{attribute 'linkalways'} 
{attribute 'no_explicit_call' := 'This FB is a CLASS and must be accessed using methods or properties'}
{attribute 'enable_dynamic_creation'}
FUNCTION_BLOCK _TIMESTRUCT EXTENDS StructuredDatatypeBase
VAR
	localData : TIMESTRUCT;
	activeData : REFERENCE TO TIMESTRUCT REF= localData;
	_wYear : _WORD(localData.wYear);
	_wMonth : _WORD(localData.wMonth);
	_wDayOfWeek : _WORD(localData.wDayOfWeek);
	_wDay : _WORD(localData.wDay);
	_wHour : _WORD(localData.wHour);
	_wMinute : _WORD(localData.wMinute);
	_wSecond : _WORD(localData.wSecond);
	_wMilliseconds : _WORD(localData.wMilliseconds);
END_VAR

PROPERTY PUBLIC Address : PVOID
GET
Address := ADR(activeData);
END_GET
END_PROPERTY

METHOD PUBLIC ClearReference
VAR_INPUT
END_VAR
activeData REF= localData;
SetMemberReference();
END_METHOD

METHOD PUBLIC Clone : I_Datatype
VAR
    pClone : POINTER TO _TIMESTRUCT;
END_VAR
pClone := __NEW(_TIMESTRUCT());
pClone^.Value := Value;
Clone := pClone^;
END_METHOD

METHOD FB_init : BOOL
VAR_INPUT
	bInitRetains : BOOL; // if TRUE, the retain variables are initialized (warm start / cold start)
	bInCopyCode : BOOL;  // if TRUE, the instance afterwards gets moved into the copy code (online change)
END_VAR
SetMemberReference();
AddMember('wYear',_wYear);
AddMember('wMonth',_wMonth);
AddMember('wDayOfWeek',_wDayOfWeek);
AddMember('wDay',_wDay);
AddMember('wHour',_wHour);
AddMember('wMinute',_wMinute);
AddMember('wSecond',_wSecond);
AddMember('wMilliseconds',_wMilliseconds);
END_METHOD

PROPERTY PUBLIC Identifier : T_MAXSTRING
GET
Identifier := 'TIMESTRUCT';
END_GET
END_PROPERTY

METHOD PUBLIC MakeReferenceTo
VAR_INPUT
	ReferenceTarget : REFERENCE TO TIMESTRUCT;
END_VAR
activeData REF= ReferenceTarget;
SetMemberReference();
END_METHOD

METHOD PROTECTED SetMemberReference
VAR_INPUT
END_VAR
_wYear.MakeReferenceTo(activeData.wYear);
_wMonth.MakeReferenceTo(activeData.wMonth);
_wDayOfWeek.MakeReferenceTo(activeData.wDayOfWeek);
_wDay.MakeReferenceTo(activeData.wDay);
_wHour.MakeReferenceTo(activeData.wHour);
_wMinute.MakeReferenceTo(activeData.wMinute);
_wSecond.MakeReferenceTo(activeData.wSecond);
_wMilliseconds.MakeReferenceTo(activeData.wMilliseconds);
END_METHOD

PROPERTY PUBLIC Size : UDINT
GET
Size := SIZEOF(activeData);
END_GET
END_PROPERTY

METHOD TryMakeReferenceTo : BOOL
VAR_INPUT
	Target : I_Datatype;
END_VAR
VAR
	pTargetData : POINTER TO TIMESTRUCT;
END_VAR
IF NOT (Target.TypeName = TypeName) THEN
	RETURN;
END_IF

pTargetData := Target.Address;
activeData REF= pTargetData^;
SetMemberReference();
TryMakeReferenceTo := TRUE;
END_METHOD

PROPERTY PUBLIC Value : REFERENCE TO TIMESTRUCT
GET
Value REF= activeData;
END_GET
END_PROPERTY

PROPERTY PUBLIC wDay : Reference to _WORD
GET
wDay REF= _wDay;
END_GET
END_PROPERTY

PROPERTY PUBLIC wDayOfWeek : Reference to _WORD
GET
wDayOfWeek REF= _wDayOfWeek;
END_GET
END_PROPERTY

PROPERTY PUBLIC wHour : Reference to _WORD
GET
wHour REF= _wHour;
END_GET
END_PROPERTY

PROPERTY PUBLIC wMilliseconds : Reference to _WORD
GET
wMilliseconds REF= _wMilliseconds;
END_GET
END_PROPERTY

PROPERTY PUBLIC wMinute : Reference to _WORD
GET
wMinute REF= _wMinute;
END_GET
END_PROPERTY

PROPERTY PUBLIC wMonth : Reference to _WORD
GET
wMonth REF= _wMonth;
END_GET
END_PROPERTY

PROPERTY PUBLIC wSecond : Reference to _WORD
GET
wSecond REF= _wSecond;
END_GET
END_PROPERTY

PROPERTY PUBLIC wYear : Reference to _WORD
GET
wYear REF= _wYear;
END_GET
END_PROPERTY

END_FUNCTION_BLOCK

(* stored: Version 1.1.0.1, ProductVersion 3.1.4024.12
   POU _TIMESTRUCT: Id {e562b4d5-1171-0283-3cd5-573928ea5f08}, SpecialFunc None
   Folder Constructor: Id {a76fe964-4813-0dcc-3a87-52590a5beee4}
   Folder Protected: Id {b9713e34-49dc-0c25-27b9-d826f124e7e3}
   Property Address: Id {bb392fc3-3f0a-0e40-3700-c5663ef20063}
   Get Get: Id {6c22c66d-e36f-0aa4-2e36-5137ed472e2a}
   Method ClearReference: Id {2cb1a7a5-525f-094b-192a-13a283037e83}
   Method Clone: Id {351d97c3-851a-0daa-253f-1e9867ba5cc1}
   Method FB_init: Id {de249045-14c0-0c8e-3c32-9e332517c285}
   Property Identifier: Id {320cbb58-8004-0152-2111-dbc950bf6d4d}
   Get Get: Id {22f478c1-48ff-0d8c-1e28-359278e8bec7}
   Method MakeReferenceTo: Id {212e5344-3a4d-0d8c-22d5-17c348eff1df}
   Method SetMemberReference: Id {153ff1cd-4750-0dd7-22e7-155c91555b63}
   Property Size: Id {212b9de1-90be-01f3-0673-9ded294ddc75}
   Get Get: Id {541f10ed-fb82-0760-3537-2ccba0ff1404}
   Method TryMakeReferenceTo: Id {436cbb68-52af-07f8-1875-c0f6af217281}
   Property Value: Id {aae5b600-b6e3-0a73-2071-e343a31d09f7}
   Get Get: Id {595b6fc1-b502-08e3-2f56-be28310fd013}
   Property wDay: Id {bdfde783-bbe0-0f05-2fda-747386cce035}
   Get Get: Id {2ff1f2ca-f10f-022c-12ce-cb56c90848c2}
   Property wDayOfWeek: Id {b3a7e28e-5e16-0746-0099-3fb50c70e777}
   Get Get: Id {f945a899-5b24-0781-3fef-24a9bc7b1ba0}
   Property wHour: Id {91565ed2-d330-0a7e-029e-facc5a7353e9}
   Get Get: Id {0672e413-fccd-0ef3-08cb-16aef2b34fd1}
   Property wMilliseconds: Id {9bf32d92-8c98-07f4-25c8-2d263c2e8511}
   Get Get: Id {ae5e8915-e489-039a-29fa-4de80ddbf57b}
   Property wMinute: Id {eed4cd1f-750b-0370-146a-dd8fe50b813b}
   Get Get: Id {4e73a3f3-2a8c-07c4-18aa-47c3230d9fee}
   Property wMonth: Id {d96efd92-1a68-076b-05e4-58cd4947e090}
   Get Get: Id {ed0b569c-4b98-0032-1e14-b67eb11dcc84}
   Property wSecond: Id {e04a2f03-75e0-017e-0a3c-599b1fc68072}
   Get Get: Id {6693ddd6-0041-0cf1-28c4-85d4dba95088}
   Property wYear: Id {078594f1-8bdb-0fe3-398d-a39a54b63005}
   Get Get: Id {127c4742-51e2-07ee-030e-9d54b8131862} *)
